// TIA Portal V18 export
// export: Created 2025-12-01T12:38:53.6836452Z, ExportSetting None, DisplayName Totally Integrated Automation Portal, DisplayVersion V18 Update 5, DisplayName TIA Portal Openness, DisplayVersion V18 Update 5, DisplayName TIA Portal Teamcenter Gateway, DisplayVersion V18, DisplayName TIA Portal Version Control Interface, DisplayVersion V18, DisplayName STEP 7 Professional, DisplayVersion V18 Update 5, DisplayName STEP 7 Safety, DisplayVersion V18, DisplayName WinCC Professional, DisplayVersion V18 Update 5
DATA_BLOCK "MES_CHeck_DB"   // DB111
// stored: AutoNumber false, InstanceOfName MES_CHeck, InstanceOfType FB
"MES_CHeck"
   // VAR
   //    Station_1 : "MES Check_fb";
   //    Station_2 : "MES Check_fb";
   //    Station_3 : "MES Check_fb";
   //    Station_4 : "MES Check_fb";
   //    Station_5 : "MES Check_fb";
   //    Station_6 : "MES Check_fb";
   //    Station_7 : "MES Check_fb";
   //    Station_8 : "MES Check_fb";
   // END_VAR
BEGIN
END_DATA_BLOCK
